# B&R Automation Studio project CleanChemi_SiteManagementSystem (part 21)

#### CMD.st
```iecst
ACTION Modbus_CMD_action:

	// --------------------------------------------------------------------
	// Variable Write Commands
	// --------------------------------------------------------------------

	// AS Block 12 - UNIT_ID
	IF gCMD_LR[IdxSkids_LR].Write_UNIT_ID.Send THEN
		MasterConfig_LR[IdxSkids_LR].action_enable[11].single := TRUE;
		gCMD_LR[IdxSkids_LR].Write_UNIT_ID.Send := FALSE;
	END_IF;

	// AS Block 13 - P201_STRT_CMD
	IF gCMD_LR[IdxSkids_LR].Write_P201_STRT_CMD.Send THEN
		MasterConfig_LR[IdxSkids_LR].action_enable[12].single := TRUE;
		gCMD_LR[IdxSkids_LR].Write_P201_STRT_CMD.Send := FALSE;
	END_IF;

	// AS Block 14 - P201_STP_CMD
	IF gCMD_LR[IdxSkids_LR].Write_P201_STP_CMD.Send THEN
		MasterConfig_LR[IdxSkids_LR].action_enable[13].single := TRUE;
		gCMD_LR[IdxSkids_LR].Write_P201_STP_CMD.Send := FALSE;
	END_IF;

	// AS Block 15 - P201_HOA
	IF gCMD_LR[IdxSkids_LR].Write_P201_HOA.Send THEN
		gCMD_LR[IdxSkids_LR].Write_P201_HOA.wP201_HOA := STRING_TO_UINT(gCMD_LR[IdxSkids_LR].Write_P201_HOA.wP201_HOA_String);
		MasterConfig_LR[IdxSkids_LR].action_enable[14].single := TRUE;
		gCMD_LR[IdxSkids_LR].Write_P201_HOA.Send := FALSE;
	ELSIF NOT gVis.Main.Out.DialogOpen THEN
		gCMD_LR[IdxSkids_LR].Write_P201_HOA.wP201_HOA_String := UINT_TO_STRING(gSkid_LR[IdxSkids_LR].Dosing_Pump_201.P201_HOA);
	END_IF;

	// AS Block 16 - P201_PPM
	IF gCMD_LR[IdxSkids_LR].Write_P201_PPM.Send THEN
		gCMD_LR[IdxSkids_LR].Write_P201_PPM.wP201_PPM_SWAPPED := IDEC_REAL_Conv(gCMD_LR[IdxSkids_LR].Write_P201_PPM.wP201_PPM);
		MasterConfig_LR[IdxSkids_LR].action_enable[15].single := TRUE;
		gCMD_LR[IdxSkids_LR].Write_P201_PPM.Send := FALSE;
	END_IF;

	// AS Block 17 - P201_SP
	IF gCMD_LR[IdxSkids_LR].Write_P201_SP.Send THEN
		gCMD_LR[IdxSkids_LR].Write_P201_SP.wP201_SP_SWAPPED := IDEC_REAL_Conv(gCMD_LR[IdxSkids_LR].Write_P201_SP.wP201_SP);
		MasterConfig_LR[IdxSkids_LR].action_enable[16].single := TRUE;
		gCMD_LR[IdxSkids_LR].Write_P201_SP.Send := FALSE;
	END_IF;

	// AS Block 18 - P202_STRT_CMD
	IF gCMD_LR[IdxSkids_LR].Write_P202_STRT_CMD.Send THEN
		MasterConfig_LR[IdxSkids_LR].action_enable[17].single := TRUE;
		gCMD_LR[IdxSkids_LR].Write_P202_STRT_CMD.Send := FALSE;
	END_IF;

	// AS Block 19 - P202_STP_CMD
	IF gCMD_LR[IdxSkids_LR].Write_P202_STP_CMD.Send THEN
		MasterConfig_LR[IdxSkids_LR].action_enable[18].single := TRUE;
		gCMD_LR[IdxSkids_LR].Write_P202_STP_CMD.Send := FALSE;
	END_IF;

	// AS Block 20 - P202_HOA
	IF gCMD_LR[IdxSkids_LR].Write_P202_HOA.Send THEN
		gCMD_LR[IdxSkids_LR].Write_P202_HOA.wP202_HOA := STRING_TO_UINT(gCMD_LR[IdxSkids_LR].Write_P202_HOA.wP202_HOA_String);
		MasterConfig_LR[IdxSkids_LR].action_enable[19].single := TRUE;
		gCMD_LR[IdxSkids_LR].Write_P202_HOA.Send := FALSE;
	ELSIF NOT gVis.Main.Out.DialogOpen THEN
		gCMD_LR[IdxSkids_LR].Write_P202_HOA.wP202_HOA_String := UINT_TO_STRING(gSkid_LR[IdxSkids_LR].Dosing_Pump_202.P202_HOA);
	END_IF;

	// AS Block 21 - P202_PPM
	IF gCMD_LR[IdxSkids_LR].Write_P202_PPM.Send THEN
		gCMD_LR[IdxSkids_LR].Write_P202_PPM.wP202_PPM_SWAPPED := IDEC_REAL_Conv(gCMD_LR[IdxSkids_LR].Write_P202_PPM.wP202_PPM);
		MasterConfig_LR[IdxSkids_LR].action_enable[20].single := TRUE;
		gCMD_LR[IdxSkids_LR].Write_P202_PPM.Send := FALSE;
	END_IF;

	// AS Block 22 - P202_SP
	IF gCMD_LR[IdxSkids_LR].Write_P202_SP.Send THEN
		gCMD_LR[IdxSkids_LR].Write_P202_SP.wP202_SP_SWAPPED := IDEC_REAL_Conv(gCMD_LR[IdxSkids_LR].Write_P202_SP.wP202_SP);
		MasterConfig_LR[IdxSkids_LR].action_enable[21].single := TRUE;
		gCMD_LR[IdxSkids_LR].Write_P202_SP.Send := FALSE;
	END_IF;

	// AS Block 23 - P203_STRT_CMD
	IF gCMD_LR[IdxSkids_LR].Write_P203_STRT_CMD.Send THEN
		MasterConfig_LR[IdxSkids_LR].action_enable[22].single := TRUE;
		gCMD_LR[IdxSkids_LR].Write_P203_STRT_CMD.Send := FALSE;
	END_IF;

	// AS Block 24 - P203_STP_CMD
	IF gCMD_LR[IdxSkids_LR].Write_P203_STP_CMD.Send THEN
		MasterConfig_LR[IdxSkids_LR].action_enable[23].single := TRUE;
		gCMD_LR[IdxSkids_LR].Write_P203_STP_CMD.Send := FALSE;
	END_IF;

	// AS Block 25 - P203_HOA
	IF gCMD_LR[IdxSkids_LR].Write_P203_HOA.Send THEN
		gCMD_LR[IdxSkids_LR].Write_P203_HOA.wP203_HOA := STRING_TO_UINT(gCMD_LR[IdxSkids_LR].Write_P203_HOA.wP203_HOA_String);
		MasterConfig_LR[IdxSkids_LR].action_enable[24].single := TRUE;
		gCMD_LR[IdxSkids_LR].Write_P203_HOA.Send := FALSE;
	ELSIF NOT gVis.Main.Out.DialogOpen THEN
		gCMD_LR[IdxSkids_LR].Write_P203_HOA.wP203_HOA_String := UINT_TO_STRING(gSkid_LR[IdxSkids_LR].Dosing_Pump_203.P203_HOA);
	END_IF;

	// AS Block 26 - P203_PPM
	IF gCMD_LR[IdxSkids_LR].Write_P203_PPM.Send THEN
		gCMD_LR[IdxSkids_LR].Write_P203_PPM.wP203_PPM_SWAPPED := IDEC_REAL_Conv(gCMD_LR[IdxSkids_LR].Write_P203_PPM.wP203_PPM);
		MasterConfig_LR[IdxSkids_LR].action_enable[25].single := TRUE;
		gCMD_LR[IdxSkids_LR].Write_P203_PPM.Send := FALSE;
	END_IF;

	// AS Block 27 - P203_SP
	IF gCMD_LR[IdxSkids_LR].Write_P203_SP.Send THEN
		gCMD_LR[IdxSkids_LR].Write_P203_SP.wP203_SP_SWAPPED := IDEC_REAL_Conv(gCMD_LR[IdxSkids_LR].Write_P203_SP.wP203_SP);
		MasterConfig_LR[IdxSkids_LR].action_enable[26].single := TRUE;
		gCMD_LR[IdxSkids_LR].Write_P203_SP.Send := FALSE;
	END_IF;

	// AS Block 28 - EFF_1
	IF gCMD_LR[IdxSkids_LR].Write_EFF_1.Send THEN
		gCMD_LR[IdxSkids_LR].Write_EFF_1.wEFF_1_SWAPPED := IDEC_REAL_Conv(gCMD_LR[IdxSkids_LR].Write_EFF_1.wEFF_1);
		MasterConfig_LR[IdxSkids_LR].action_enable[27].single := TRUE;
		gCMD_LR[IdxSkids_LR].Write_EFF_1.Send := FALSE;
	END_IF;

	// AS Block 29 - EFF_2
	IF gCMD_LR[IdxSkids_LR].Write_EFF_2.Send THEN
		gCMD_LR[IdxSkids_LR].Write_EFF_2.wEFF_2_SWAPPED := IDEC_REAL_Conv(gCMD_LR[IdxSkids_LR].Write_EFF_2.wEFF_2);
		MasterConfig_LR[IdxSkids_LR].action_enable[28].single := TRUE;
		gCMD_LR[IdxSkids_LR].Write_EFF_2.Send := FALSE;
	END_IF;

	// AS Block 30 - NAOH_TO_H2O2
	IF gCMD_LR[IdxSkids_LR].Write_NAOH_TO_H2O2.Send THEN
		gCMD_LR[IdxSkids_LR].Write_NAOH_TO_H2O2.wNAOH_TO_H2O2_SWAPPED := IDEC_REAL_Conv(gCMD_LR[IdxSkids_LR].Write_NAOH_TO_H2O2.wNAOH_TO_H2O2);
		MasterConfig_LR[IdxSkids_LR].action_enable[29].single := TRUE;
		gCMD_LR[IdxSkids_LR].Write_NAOH_TO_H2O2.Send := FALSE;
	END_IF;

	// AS Block 31 - TRI_TO_H2O2
	IF gCMD_LR[IdxSkids_LR].Write_TRI_TO_H2O2.Send THEN
		gCMD_LR[IdxSkids_LR].Write_TRI_TO_H2O2.wTRI_TO_H2O2_SWAPPED := IDEC_REAL_Conv(gCMD_LR[IdxSkids_LR].Write_TRI_TO_H2O2.wTRI_TO_H2O2);
		MasterConfig_LR[IdxSkids_LR].action_enable[30].single := TRUE;
		gCMD_LR[IdxSkids_LR].Write_TRI_TO_H2O2.Send := FALSE;
	END_IF;

	// AS Block 32 - PMAX_HOA
	IF gCMD_LR[IdxSkids_LR].Write_PMAX_HOA.Send THEN
		gCMD_LR[IdxSkids_LR].Write_PMAX_HOA.wPMAX_HOA := STRING_TO_UINT(gCMD_LR[IdxSkids_LR].Write_PMAX_HOA.wPMAX_HOA_String);
		MasterConfig_LR[IdxSkids_LR].action_enable[31].single := TRUE;
		gCMD_LR[IdxSkids_LR].Write_PMAX_HOA.Send := FALSE;
	ELSIF NOT gVis.Main.Out.DialogOpen THEN
		gCMD_LR[IdxSkids_LR].Write_PMAX_HOA.wPMAX_HOA_String := UINT_TO_STRING(gSkid_LR[IdxSkids_LR].Pmax_General_Variables.PMAX_HOA);
	END_IF;

	// AS Block 33 - PMAX_CONC
	IF gCMD_LR[IdxSkids_LR].Write_PMAX_CONC.Send THEN
		gCMD_LR[IdxSkids_LR].Write_PMAX_CONC.wPMAX_CONC_SWAPPED := IDEC_REAL_Conv(gCMD_LR[IdxSkids_LR].Write_PMAX_CONC.wPMAX_CONC);
		MasterConfig_LR[IdxSkids_LR].action_enable[32].single := TRUE;
		gCMD_LR[IdxSkids_LR].Write_PMAX_CONC.Send := FALSE;
	END_IF;

	// AS Block 34 - HP_CONC
	IF gCMD_LR[IdxSkids_LR].Write_HP_CONC.Send THEN
		gCMD_LR[IdxSkids_LR].Write_HP_CONC.wHP_CONC_SWAPPED := IDEC_REAL_Conv(gCMD_LR[IdxSkids_LR].Write_HP_CONC.wHP_CONC);
		MasterConfig_LR[IdxSkids_LR].action_enable[33].single := TRUE;
		gCMD_LR[IdxSkids_LR].Write_HP_CONC.Send := FALSE;
	END_IF;

	// AS Block 35 - NAOH_CONC
	IF gCMD_LR[IdxSkids_LR].Write_NAOH_CONC.Send THEN
		gCMD_LR[IdxSkids_LR].Write_NAOH_CONC.wNAOH_CONC_SWAPPED := IDEC_REAL_Conv(gCMD_LR[IdxSkids_LR].Write_NAOH_CONC.wNAOH_CONC);
		MasterConfig_LR[IdxSkids_LR].action_enable[34].single := TRUE;
		gCMD_LR[IdxSkids_LR].Write_NAOH_CONC.Send := FALSE;
	END_IF;

	// AS Block 36 - P101_STRT_CMD
	IF gCMD_LR[IdxSkids_LR].Write_P101_STRT_CMD.Send THEN
		MasterConfig_LR[IdxSkids_LR].action_enable[35].single := TRUE;
		gCMD_LR[IdxSkids_LR].Write_P101_STRT_CMD.Send := FALSE;
	END_IF;

	// AS Block 37 - P101_STP_CMD
	IF gCMD_LR[IdxSkids_LR].Write_P101_STP_CMD.Send THEN
		MasterConfig_LR[IdxSkids_LR].action_enable[36].single := TRUE;
		gCMD_LR[IdxSkids_LR].Write_P101_STP_CMD.Send := FALSE;
	END_IF;

	// AS Block 38 - P101_SP
	IF gCMD_LR[IdxSkids_LR].Write_P101_SP.Send THEN
		gCMD_LR[IdxSkids_LR].Write_P101_SP.wP101_SP_SWAPPED := IDEC_REAL_Conv(gCMD_LR[IdxSkids_LR].Write_P101_SP.wP101_SP);
		MasterConfig_LR[IdxSkids_LR].action_enable[37].single := TRUE;
		gCMD_LR[IdxSkids_LR].Write_P101_SP.Send := FALSE;
	END_IF;

	// AS Block 39 - P102_STRT_CMD
	IF gCMD_LR[IdxSkids_LR].Write_P102_STRT_CMD.Send THEN
		MasterConfig_LR[IdxSkids_LR].action_enable[38].single := TRUE;
		gCMD_LR[IdxSkids_LR].Write_P102_STRT_CMD.Send := FALSE;
	END_IF;

	// AS Block 40 - P102_STP_CMD
	IF gCMD_LR[IdxSkids_LR].Write_P102_STP_CMD.Send THEN
		MasterConfig_LR[IdxSkids_LR].action_enable[39].single := TRUE;
		gCMD_LR[IdxSkids_LR].Write_P102_STP_CMD.Send := FALSE;
	END_IF;

	// AS Block 41 - P102_SP
	IF gCMD_LR[IdxSkids_LR].Write_P102_SP.Send THEN
		gCMD_LR[IdxSkids_LR].Write_P102_SP.wP102_SP_SWAPPED := IDEC_REAL_Conv(gCMD_LR[IdxSkids_LR].Write_P102_SP.wP102_SP);
		MasterConfig_LR[IdxSkids_LR].action_enable[40].single := TRUE;
		gCMD_LR[IdxSkids_LR].Write_P102_SP.Send := FALSE;
	END_IF;

	// AS Block 42 - P103_STRT_CMD
	IF gCMD_LR[IdxSkids_LR].Write_P103_STRT_CMD.Send THEN
		MasterConfig_LR[IdxSkids_LR].action_enable[41].single := TRUE;
		gCMD_LR[IdxSkids_LR].Write_P103_STRT_CMD.Send := FALSE;
	END_IF;

	// AS Block 43 - P103_STP_CMD
	IF gCMD_LR[IdxSkids_LR].Write_P103_STP_CMD.Send THEN
		MasterConfig_LR[IdxSkids_LR].action_enable[42].single := TRUE;
		gCMD_LR[IdxSkids_LR].Write_P103_STP_CMD.Send := FALSE;
	END_IF;

	// AS Block 44 - P103_SP
	IF gCMD_LR[IdxSkids_LR].Write_P103_SP.Send THEN
		gCMD_LR[IdxSkids_LR].Write_P103_SP.wP103_SP_SWAPPED := IDEC_REAL_Conv(gCMD_LR[IdxSkids_LR].Write_P103_SP.wP103_SP);
		MasterConfig_LR[IdxSkids_LR].action_enable[43].single := TRUE;
		gCMD_LR[IdxSkids_LR].Write_P103_SP.Send := FALSE;
	END_IF;

	// AS Block 45 - P104_STRT_CMD
	IF gCMD_LR[IdxSkids_LR].Write_P104_STRT_CMD.Send THEN
		MasterConfig_LR[IdxSkids_LR].action_enable[44].single := TRUE;
		gCMD_LR[IdxSkids_LR].Write_P103_STRT_CMD.Send := FALSE;
	END_IF;

	// AS Block 46 - P104_STP_CMD
	IF gCMD_LR[IdxSkids_LR].Write_P104_STP_CMD.Send THEN
		MasterConfig_LR[IdxSkids_LR].action_enable[45].single := TRUE;
		gCMD_LR[IdxSkids_LR].Write_P104_STP_CMD.Send := FALSE;
	END_IF;

	// AS Block 47 - P104_SP
	IF gCMD_LR[IdxSkids_LR].Write_P104_SP.Send THEN
		gCMD_LR[IdxSkids_LR].Write_P104_SP.wP104_SP_SWAPPED := IDEC_REAL_Conv(gCMD_LR[IdxSkids_LR].Write_P104_SP.wP104_SP);
		MasterConfig_LR[IdxSkids_LR].action_enable[46].single := TRUE;
		gCMD_LR[IdxSkids_LR].Write_P104_SP.Send := FALSE;
	END_IF;

	// AS Block 48 is a READ block

	// AS Block 49 - LOCK_CMD
	IF gCMD_LR[IdxSkids_LR].Write_LOCK_CMD.Send THEN
		MasterConfig_LR[IdxSkids_LR].action_enable[48].single := TRUE;
		gCMD_LR[IdxSkids_LR].Write_LOCK_CMD.Send := FALSE;
	END_IF;

	// AS Block 50 - UNLOCK_CMD
	IF gCMD_LR[IdxSkids_LR].Write_UNLOCK_CMD.Send THEN
		MasterConfig_LR[IdxSkids_LR].action_enable[49].single := TRUE;
		gCMD_LR[IdxSkids_LR].Write_UNLOCK_CMD.Send := FALSE;
	END_IF;

	// AS Block 51 - FI301_SIM_CMD
	IF gCMD_LR[IdxSkids_LR].Write_FI301_SIM_CMD.Send THEN
		MasterConfig_LR[IdxSkids_LR].action_enable[50].single := TRUE;
		gCMD_LR[IdxSkids_LR].Write_FI301_SIM_CMD.Send := FALSE;
	END_IF;

	// AS Block 52 - FI301_MEA_CMD
	IF gCMD_LR[IdxSkids_LR].Write_FI301_MEA_CMD.Send THEN
		MasterConfig_LR[IdxSkids_LR].action_enable[51].single := TRUE;
		gCMD_LR[IdxSkids_LR].Write_FI301_MEA_CMD.Send := FALSE;
	END_IF;

	// AS Block 53 - FI301_SIM
	IF gCMD_LR[IdxSkids_LR].Write_FI301_SIM.Send THEN
		gCMD_LR[IdxSkids_LR].Write_FI301_SIM.wFI301_SIM_SWAPPED := IDEC_REAL_Conv(gCMD_LR[IdxSkids_LR].Write_FI301_SIM.wFI301_SIM);
		MasterConfig_LR[IdxSkids_LR].action_enable[52].single := TRUE;
		gCMD_LR[IdxSkids_LR].Write_FI301_SIM.Send := FALSE;
	END_IF;

	// AS Block 54 - FI302_SIM_CMD
	IF gCMD_LR[IdxSkids_LR].Write_FI302_SIM_CMD.Send THEN
		MasterConfig_LR[IdxSkids_LR].action_enable[53].single := TRUE;
		gCMD_LR[IdxSkids_LR].Write_FI302_SIM_CMD.Send := FALSE;
	END_IF;

	// AS Block 55 - FI302_MEA_CMD
	IF gCMD_LR[IdxSkids_LR].Write_FI302_MEA_CMD.Send THEN
		MasterConfig_LR[IdxSkids_LR].action_enable[54].single := TRUE;
		gCMD_LR[IdxSkids_LR].Write_FI302_MEA_CMD.Send := FALSE;
	END_IF;

	// AS Block 56 - FI302_SIM
	IF gCMD_LR[IdxSkids_LR].Write_FI302_SIM.Send THEN
		gCMD_LR[IdxSkids_LR].Write_FI302_SIM.wFI302_SIM_SWAPPED := IDEC_REAL_Conv(gCMD_LR[IdxSkids_LR].Write_FI302_SIM.wFI302_SIM);
		MasterConfig_LR[IdxSkids_LR].action_enable[55].single := TRUE;
		gCMD_LR[IdxSkids_LR].Write_FI302_SIM.Send := FALSE;
	END_IF;

	// AS Block 57 - FI303_SIM_CMD
	IF gCMD_LR[IdxSkids_LR].Write_FI303_SIM_CMD.Send THEN
		MasterConfig_LR[IdxSkids_LR].action_enable[56].single := TRUE;
		gCMD_LR[IdxSkids_LR].Write_FI303_SIM_CMD.Send := FALSE;
	END_IF;

	// AS Block 58 - FI303_MEA_CMD
	IF gCMD_LR[IdxSkids_LR].Write_FI303_MEA_CMD.Send THEN
		MasterConfig_LR[IdxSkids_LR].action_enable[57].single := TRUE;
		gCMD_LR[IdxSkids_LR].Write_FI303_MEA_CMD.Send := FALSE;
	END_IF;

	// AS Block 59 - FI303_SIM
	IF gCMD_LR[IdxSkids_LR].Write_FI303_SIM.Send THEN
		gCMD_LR[IdxSkids_LR].Write_FI303_SIM.wFI303_SIM_SWAPPED := IDEC_REAL_Conv(gCMD_LR[IdxSkids_LR].Write_FI303_SIM.wFI303_SIM);
		MasterConfig_LR[IdxSkids_LR].action_enable[58].single := TRUE;
		gCMD_LR[IdxSkids_LR].Write_FI303_SIM.Send := FALSE;
	END_IF;

	// AS Block 60 - UNIT_ACK - RESET OF CONDITION PERFORMED IN MAIN.ST ALARMS RESET
	IF gVis.Main.In.AckAllAlarms_Skid[IdxSkids_LR] THEN
		MasterConfig_LR[IdxSkids_LR].action_enable[59].single := TRUE;
	END_IF;

	// AS Block 61 IS THE TEXT READ INT BLOCK

	// AS Block 62 - XV101_OPEN_CMD
	IF gCMD_LR[IdxSkids_LR].Write_XV101_OPEN_CMD.Send THEN
		MasterConfig_LR[IdxSkids_LR].action_enable[61].single := TRUE;
		gCMD_LR[IdxSkids_LR].Write_XV101_OPEN_CMD.Send := FALSE;
	END_IF;

	// AS Block 63 - XV102_OPEN_CMD
	IF gCMD_LR[IdxSkids_LR].Write_XV102_OPEN_CMD.Send THEN
		MasterConfig_LR[IdxSkids_LR].action_enable[62].single := TRUE;
		gCMD_LR[IdxSkids_LR].Write_XV102_OPEN_CMD.Send := FALSE;
	END_IF;

	// AS Block 64 - XV103_OPEN_CMD
	IF gCMD_LR[IdxSkids_LR].Write_XV103_OPEN_CMD.Send THEN
		MasterConfig_LR[IdxSkids_LR].action_enable[63].single := TRUE;
		gCMD_LR[IdxSkids_LR].Write_XV103_OPEN_CMD.Send := FALSE;
	END_IF;

	// AS Block 65 - XV104_OPEN_CMD
	IF gCMD_LR[IdxSkids_LR].Write_XV104_OPEN_CMD.Send THEN
		MasterConfig_LR[IdxSkids_LR].action_enable[64].single := TRUE;
		gCMD_LR[IdxSkids_LR].Write_XV104_OPEN_CMD.Send := FALSE;
	END_IF;

	// AS Block 66 - XV201_OPEN_CMD
	IF gCMD_LR[IdxSkids_LR].Write_XV201_OPEN_CMD.Send THEN
		MasterConfig_LR[IdxSkids_LR].action_enable[65].single := TRUE;
		gCMD_LR[IdxSkids_LR].Write_XV201_OPEN_CMD.Send := FALSE;
	END_IF;

	// AS Block 67 - XV202_OPEN_CMD
	IF gCMD_LR[IdxSkids_LR].Write_XV202_OPEN_CMD.Send THEN
		MasterConfig_LR[IdxSkids_LR].action_enable[66].single := TRUE;
		gCMD_LR[IdxSkids_LR].Write_XV202_OPEN_CMD.Send := FALSE;
	END_IF;

	// AS Block 68 - XV203_OPEN_CMD
	IF gCMD_LR[IdxSkids_LR].Write_XV203_OPEN_CMD.Send THEN
		MasterConfig_LR[IdxSkids_LR].action_enable[67].single := TRUE;
		gCMD_LR[IdxSkids_LR].Write_XV203_OPEN_CMD.Send := FALSE;
	END_IF;

	// AS Block 69 - AS_USER
	IF gCMD_LR[IdxSkids_LR].Write_AS_USER.Send THEN
		MasterConfig_LR[IdxSkids_LR].action_enable[68].single := TRUE;
		gCMD_LR[IdxSkids_LR].Write_AS_USER.Send := FALSE;
	END_IF;

	// AS Block 70 - AS_ACCESS
	IF gCMD_LR[IdxSkids_LR].Write_AS_ACCESS.Send THEN
		MasterConfig_LR[IdxSkids_LR].action_enable[69].single := TRUE;
		gCMD_LR[IdxSkids_LR].Write_AS_ACCESS.Send := FALSE;
	END_IF;

	// AS Block 71 - TOTALIZER_RESET
	IF gCMD_LR[IdxSkids_LR].Write_TOTALIZER_RESET.Send THEN
		MasterConfig_LR[IdxSkids_LR].action_enable[70].single := TRUE;
		gCMD_LR[IdxSkids_LR].Write_TOTALIZER_RESET.Send := FALSE;
	END_IF;

END_ACTION
```

#### Status.st
```iecst
ACTION Modbus_Status_action:

	ModbusTcpMaster[IdxSkids_LR]();

	// --------------------------------------------------------------------
	// Reset last error information
	// --------------------------------------------------------------------
	IF(reset_error) THEN
		brsmemset(ADR(ModbusTcpMaster[IdxSkids_LR].last_error), 0, 2);
		reset_error := 0;
	END_IF

	// --------------------------------------------------------------------
	// Final Variable Mapping AND Data Conversion - READ
	// --------------------------------------------------------------------

	// force transfer
	// AS Block 1 - 6000 DOSING INT
	gSkid_LR[IdxSkids_LR].Pmax_General_Variables.UNIT_ID := gModbus_LR[IdxSkids_LR].Modbus_PeroxyMAX.Block1_Int[0];
	gSkid_LR[IdxSkids_LR].Pmax_General_Variables.USER_ID := gModbus_LR[IdxSkids_LR].Modbus_PeroxyMAX.Block1_Int[2];
	gSkid_LR[IdxSkids_LR].Pmax_General_Variables.USER_ACCESS := gModbus_LR[IdxSkids_LR].Modbus_PeroxyMAX.Block1_Int[4];
	gSkid_LR[IdxSkids_LR].Pmax_General_Variables.PMAX_HOA := gModbus_LR[IdxSkids_LR].Modbus_PeroxyMAX.Block1_Int[6];
	gSkid_LR[IdxSkids_LR].Pmax_General_Variables.PMAX_STATUS := gModbus_LR[IdxSkids_LR].Modbus_PeroxyMAX.Block1_Int[8];
	gSkid_LR[IdxSkids_LR].Pmax_General_Variables.SCREEN_LOCK := gModbus_LR[IdxSkids_LR].Modbus_PeroxyMAX.Block1_Int[10];

	gSkid_LR[IdxSkids_LR].Pmax_Pump_101.P101_XS := gModbus_LR[IdxSkids_LR].Modbus_PeroxyMAX.Block1_Int[20];
	gSkid_LR[IdxSkids_LR].Sensor_Variables.XV101 := gModbus_LR[IdxSkids_LR].Modbus_PeroxyMAX.Block1_Int[22];
	gSkid_LR[IdxSkids_LR].Sensor_Variables.XV101_ENABLE := gModbus_LR[IdxSkids_LR].Modbus_PeroxyMAX.Block1_Int[24];

	gSkid_LR[IdxSkids_LR].Pmax_Pump_102.P102_XS := gModbus_LR[IdxSkids_LR].Modbus_PeroxyMAX.Block1_Int[32];
	gSkid_LR[IdxSkids_LR].Pmax_Pump_102.P102_WARN := gModbus_LR[IdxSkids_LR].Modbus_PeroxyMAX.Block1_Int[34];
	gSkid_LR[IdxSkids_LR].Pmax_Pump_102.P102_ALARM := gModbus_LR[IdxSkids_LR].Modbus_PeroxyMAX.Block1_Int[36];
	gSkid_LR[IdxSkids_LR].Sensor_Variables.XV102 := gModbus_LR[IdxSkids_LR].Modbus_PeroxyMAX.Block1_Int[38];

	gSkid_LR[IdxSkids_LR].Pmax_Pump_103.P103_XS := gModbus_LR[IdxSkids_LR].Modbus_PeroxyMAX.Block1_Int[48];
	gSkid_LR[IdxSkids_LR].Pmax_Pump_103.P103_WARN := gModbus_LR[IdxSkids_LR].Modbus_PeroxyMAX.Block1_Int[50];
	gSkid_LR[IdxSkids_LR].Pmax_Pump_103.P103_ALARM := gModbus_LR[IdxSkids_LR].Modbus_PeroxyMAX.Block1_Int[52];
	gSkid_LR[IdxSkids_LR].Sensor_Variables.XV103 := gModbus_LR[IdxSkids_LR].Modbus_PeroxyMAX.Block1_Int[54];

	gSkid_LR[IdxSkids_LR].Pmax_Pump_104.P104_XS := gModbus_LR[IdxSkids_LR].Modbus_PeroxyMAX.Block1_Int[64];
	gSkid_LR[IdxSkids_LR].Pmax_Pump_104.P104_WARN := gModbus_LR[IdxSkids_LR].Modbus_PeroxyMAX.Block1_Int[66];
	gSkid_LR[IdxSkids_LR].Pmax_Pump_104.P104_ALARM := gModbus_LR[IdxSkids_LR].Modbus_PeroxyMAX.Block1_Int[68];
	gSkid_LR[IdxSkids_LR].Sensor_Variables.XV104 := gModbus_LR[IdxSkids_LR].Modbus_PeroxyMAX.Block1_Int[70];

	// AS Block 2 - 6000 DOSING INT - SPARE
	//:= gModbus_LR[IdxSkids_LR].Modbus_PeroxyMAX.Block2_Int[0];

	// AS Block 3 - 6000 DOSING REAL
	gSkid_LR[IdxSkids_LR].ConversionRatios.EFF_1:= IDEC_REAL_Conv(gModbus_LR[IdxSkids_LR].Modbus_PeroxyMAX.Block3_Real[0]);
	gSkid_LR[IdxSkids_LR].ConversionRatios.EFF_2:= IDEC_REAL_Conv(gModbus_LR[IdxSkids_LR].Modbus_PeroxyMAX.Block3_Real[1]);
	gSkid_LR[IdxSkids_LR].ConversionRatios.NAOH_TO_H2O2:= IDEC_REAL_Conv(gModbus_LR[IdxSkids_LR].Modbus_PeroxyMAX.Block3_Real[2]);
	gSkid_LR[IdxSkids_LR].ConversionRatios.TRI_TO_H2O2:= IDEC_REAL_Conv(gModbus_LR[IdxSkids_LR].Modbus_PeroxyMAX.Block3_Real[3]);
	gSkid_LR[IdxSkids_LR].ConversionRatios.NAOH_TO_TRI:= IDEC_REAL_Conv(gModbus_LR[IdxSkids_LR].Modbus_PeroxyMAX.Block3_Real[4]);

	gSkid_LR[IdxSkids_LR].Pmax_General_Variables.PMAX_CONC:= IDEC_REAL_Conv(gModbus_LR[IdxSkids_LR].Modbus_PeroxyMAX.Block3_Real[8]);
	gSkid_LR[IdxSkids_LR].Pmax_General_Variables.PMAX_RATE:= IDEC_REAL_Conv(gModbus_LR[IdxSkids_LR].Modbus_PeroxyMAX.Block3_Real[9]);
	gSkid_LR[IdxSkids_LR].Pmax_General_Variables.PMAX_PV:= IDEC_REAL_Conv(gModbus_LR[IdxSkids_LR].Modbus_PeroxyMAX.Block3_Real[10]);
	gSkid_LR[IdxSkids_LR].Pmax_General_Variables.NAOH_CONC:= IDEC_REAL_Conv(gModbus_LR[IdxSkids_LR].Modbus_PeroxyMAX.Block3_Real[11]);
	gSkid_LR[IdxSkids_LR].Pmax_General_Variables.NAOH_CONC_OD:= IDEC_REAL_Conv(gModbus_LR[IdxSkids_LR].Modbus_PeroxyMAX.Block3_Real[12]);
	gSkid_LR[IdxSkids_LR].Pmax_General_Variables.HP_CONC:= IDEC_REAL_Conv(gModbus_LR[IdxSkids_LR].Modbus_PeroxyMAX.Block3_Real[13]);
	gSkid_LR[IdxSkids_LR].Pmax_General_Variables.HP_CONC_OD:= IDEC_REAL_Conv(gModbus_LR[IdxSkids_LR].Modbus_PeroxyMAX.Block3_Real[14]);

	gSkid_LR[IdxSkids_LR].Pmax_Pump_101.P101_SP:= IDEC_REAL_Conv(gModbus_LR[IdxSkids_LR].Modbus_PeroxyMAX.Block3_Real[21]);
	gSkid_LR[IdxSkids_LR].Pmax_Pump_101.P101_PV:= IDEC_REAL_Conv(gModbus_LR[IdxSkids_LR].Modbus_PeroxyMAX.Block3_Real[22]);
	gSkid_LR[IdxSkids_LR].Pmax_Pump_101.P101_OP:= IDEC_REAL_Conv(gModbus_LR[IdxSkids_LR].Modbus_PeroxyMAX.Block3_Real[23]);
	gSkid_LR[IdxSkids_LR].Pmax_Pump_101.P101_FQ:= IDEC_REAL_Conv(gModbus_LR[IdxSkids_LR].Modbus_PeroxyMAX.Block3_Real[24]);
	gSkid_LR[IdxSkids_LR].Pmax_Pump_101.P101_TI:= IDEC_REAL_Conv(gModbus_LR[IdxSkids_LR].Modbus_PeroxyMAX.Block3_Real[25]);
	gSkid_LR[IdxSkids_LR].Pmax_Pump_101.P101_PI:= IDEC_REAL_Conv(gModbus_LR[IdxSkids_LR].Modbus_PeroxyMAX.Block3_Real[26]);
	gSkid_LR[IdxSkids_LR].Pmax_Pump_101.P101_PFI:= IDEC_REAL_Conv(gModbus_LR[IdxSkids_LR].Modbus_PeroxyMAX.Block3_Real[27]);
	gSkid_LR[IdxSkids_LR].Pmax_Pump_101.P101_LS:= IDEC_REAL_Conv(gModbus_LR[IdxSkids_LR].Modbus_PeroxyMAX.Block3_Real[28]);

	gSkid_LR[IdxSkids_LR].Pmax_Pump_101B.P101B_OP:= IDEC_REAL_Conv(gModbus_LR[IdxSkids_LR].Modbus_PeroxyMAX.Block3_Real[35]);
	gSkid_LR[IdxSkids_LR].Pmax_Pump_101B.P101B_PFI:= IDEC_REAL_Conv(gModbus_LR[IdxSkids_LR].Modbus_PeroxyMAX.Block3_Real[36]);
	gSkid_LR[IdxSkids_LR].Pmax_Pump_101B.P101B_SP:= IDEC_REAL_Conv(gModbus_LR[IdxSkids_LR].Modbus_PeroxyMAX.Block3_Real[37]);
	gSkid_LR[IdxSkids_LR].Pmax_Pump_101B.P101B_LS:= IDEC_REAL_Conv(gModbus_LR[IdxSkids_LR].Modbus_PeroxyMAX.Block3_Real[38]);

	gSkid_LR[IdxSkids_LR].Pmax_Pump_102.P102_SP:= IDEC_REAL_Conv(gModbus_LR[IdxSkids_LR].Modbus_PeroxyMAX.Block3_Real[45]);
	gSkid_LR[IdxSkids_LR].Pmax_Pump_102.P102_PV:= IDEC_REAL_Conv(gModbus_LR[IdxSkids_LR].Modbus_PeroxyMAX.Block3_Real[46]);
	gSkid_LR[IdxSkids_LR].Pmax_Pump_102.P102_OP:= IDEC_REAL_Conv(gModbus_LR[IdxSkids_LR].Modbus_PeroxyMAX.Block3_Real[47]);
	gSkid_LR[IdxSkids_LR].Pmax_Pump_102.P102_PFI:= IDEC_REAL_Conv(gModbus_LR[IdxSkids_LR].Modbus_PeroxyMAX.Block3_Real[48]);
	gSkid_LR[IdxSkids_LR].Pmax_Pump_102.P102_FQ:= IDEC_REAL_Conv(gModbus_LR[IdxSkids_LR].Modbus_PeroxyMAX.Block3_Real[49]);
	gSkid_LR[IdxSkids_LR].Pmax_Pump_102.P102_PFQ:= IDEC_REAL_Conv(gModbus_LR[IdxSkids_LR].Modbus_PeroxyMAX.Block3_Real[50]);
	gSkid_LR[IdxSkids_LR].Pmax_Pump_102.P102_PPI:= IDEC_REAL_Conv(gModbus_LR[IdxSkids_LR].Modbus_PeroxyMAX.Block3_Real[51]);
	gSkid_LR[IdxSkids_LR].Pmax_Pump_102.P102_TI:= IDEC_REAL_Conv(gModbus_LR[IdxSkids_LR].Modbus_PeroxyMAX.Block3_Real[52]);
	gSkid_LR[IdxSkids_LR].Pmax_Pump_102.P102_PI:= IDEC_REAL_Conv(gModbus_LR[IdxSkids_LR].Modbus_PeroxyMAX.Block3_Real[53]);
	gSkid_LR[IdxSkids_LR].Pmax_Pump_102.P102_LS:= IDEC_REAL_Conv(gModbus_LR[IdxSkids_LR].Modbus_PeroxyMAX.Block3_Real[54]);

	gSkid_LR[IdxSkids_LR].Pmax_Pump_103.P103_SP:= IDEC_REAL_Conv(gModbus_LR[IdxSkids_LR].Modbus_PeroxyMAX.Block3_Real[59]);
	gSkid_LR[IdxSkids_LR].Pmax_Pump_103.P103_PV:= IDEC_REAL_Conv(gModbus_LR[IdxSkids_LR].Modbus_PeroxyMAX.Block3_Real[60]);
	gSkid_LR[IdxSkids_LR].Pmax_Pump_103.P103_OP:= IDEC_REAL_Conv(gModbus_LR[IdxSkids_LR].Modbus_PeroxyMAX.Block3_Real[61]);
	gSkid_LR[IdxSkids_LR].Pmax_Pump_103.P103_PFI:= IDEC_REAL_Conv(gModbus_LR[IdxSkids_LR].Modbus_PeroxyMAX.Block3_Real[62]);

	// AS Block 4 - 6000 DOSING REAL
	gSkid_LR[IdxSkids_LR].Pmax_Pump_103.P103_FQ:= IDEC_REAL_Conv(gModbus_LR[IdxSkids_LR].Modbus_PeroxyMAX.Block4_Real[0]);
	gSkid_LR[IdxSkids_LR].Pmax_Pump_103.P103_PFQ:= IDEC_REAL_Conv(gModbus_LR[IdxSkids_LR].Modbus_PeroxyMAX.Block4_Real[1]);
	gSkid_LR[IdxSkids_LR].Pmax_Pump_103.P103_PPI:= IDEC_REAL_Conv(gModbus_LR[IdxSkids_LR].Modbus_PeroxyMAX.Block4_Real[2]);
	gSkid_LR[IdxSkids_LR].Pmax_Pump_103.P103_TI:= IDEC_REAL_Conv(gModbus_LR[IdxSkids_LR].Modbus_PeroxyMAX.Block4_Real[3]);
	gSkid_LR[IdxSkids_LR].Pmax_Pump_103.P103_PI:= IDEC_REAL_Conv(gModbus_LR[IdxSkids_LR].Modbus_PeroxyMAX.Block4_Real[4]);
	gSkid_LR[IdxSkids_LR].Pmax_Pump_103.P103_LS:= IDEC_REAL_Conv(gModbus_LR[IdxSkids_LR].Modbus_PeroxyMAX.Block4_Real[5]);

	gSkid_LR[IdxSkids_LR].Pmax_Pump_104.P104_SP:= IDEC_REAL_Conv(gModbus_LR[IdxSkids_LR].Modbus_PeroxyMAX.Block4_Real[10]);
	gSkid_LR[IdxSkids_LR].Pmax_Pump_104.P104_PV:= IDEC_REAL_Conv(gModbus_LR[IdxSkids_LR].Modbus_PeroxyMAX.Block4_Real[11]);
	gSkid_LR[IdxSkids_LR].Pmax_Pump_104.P104_OP:= IDEC_REAL_Conv(gModbus_LR[IdxSkids_LR].Modbus_PeroxyMAX.Block4_Real[12]);
	gSkid_LR[IdxSkids_LR].Pmax_Pump_104.P104_PFI:= IDEC_REAL_Conv(gModbus_LR[IdxSkids_LR].Modbus_PeroxyMAX.Block4_Real[13]);
	gSkid_LR[IdxSkids_LR].Pmax_Pump_104.P104_FQ:= IDEC_REAL_Conv(gModbus_LR[IdxSkids_LR].Modbus_PeroxyMAX.Block4_Real[14]);
	gSkid_LR[IdxSkids_LR].Pmax_Pump_104.P104_PFQ:= IDEC_REAL_Conv(gModbus_LR[IdxSkids_LR].Modbus_PeroxyMAX.Block4_Real[15]);
	gSkid_LR[IdxSkids_LR].Pmax_Pump_104.P104_PPI:= IDEC_REAL_Conv(gModbus_LR[IdxSkids_LR].Modbus_PeroxyMAX.Block4_Real[16]);
	gSkid_LR[IdxSkids_LR].Pmax_Pump_104.P104_PI:= IDEC_REAL_Conv(gModbus_LR[IdxSkids_LR].Modbus_PeroxyMAX.Block4_Real[17]);
	gSkid_LR[IdxSkids_LR].Pmax_Pump_104.P104_LS:= IDEC_REAL_Conv(gModbus_LR[IdxSkids_LR].Modbus_PeroxyMAX.Block4_Real[18]);

	gSkid_LR[IdxSkids_LR].Sensor_Variables.CD101:= IDEC_REAL_Conv(gModbus_LR[IdxSkids_LR].Modbus_PeroxyMAX.Block4_Real[24]);
	gSkid_LR[IdxSkids_LR].Sensor_Variables.CD101_SP:= IDEC_REAL_Conv(gModbus_LR[IdxSkids_LR].Modbus_PeroxyMAX.Block4_Real[25]);
	gSkid_LR[IdxSkids_LR].Sensor_Variables.CD102:= IDEC_REAL_Conv(gModbus_LR[IdxSkids_LR].Modbus_PeroxyMAX.Block4_Real[26]);
	gSkid_LR[IdxSkids_LR].Sensor_Variables.CD102_SP:= IDEC_REAL_Conv(gModbus_LR[IdxSkids_LR].Modbus_PeroxyMAX.Block4_Real[27]);
	gSkid_LR[IdxSkids_LR].Sensor_Variables.CD103:= IDEC_REAL_Conv(gModbus_LR[IdxSkids_LR].Modbus_PeroxyMAX.Block4_Real[28]);
	gSkid_LR[IdxSkids_LR].Sensor_Variables.CD103_SP:= IDEC_REAL_Conv(gModbus_LR[IdxSkids_LR].Modbus_PeroxyMAX.Block4_Real[29]);

	gSkid_LR[IdxSkids_LR].Sensor_Variables.CD101_TI:= IDEC_REAL_Conv(gModbus_LR[IdxSkids_LR].Modbus_PeroxyMAX.Block4_Real[36]);
	gSkid_LR[IdxSkids_LR].Sensor_Variables.CD102_TI:= IDEC_REAL_Conv(gModbus_LR[IdxSkids_LR].Modbus_PeroxyMAX.Block4_Real[37]);
	gSkid_LR[IdxSkids_LR].Sensor_Variables.CD103_TI:= IDEC_REAL_Conv(gModbus_LR[IdxSkids_LR].Modbus_PeroxyMAX.Block4_Real[38]);

	gSkid_LR[IdxSkids_LR].Pmax_General_Variables.HMI_REV_A:= IDEC_REAL_Conv(gModbus_LR[IdxSkids_LR].Modbus_PeroxyMAX.Block4_Real[45]);
	gSkid_LR[IdxSkids_LR].Pmax_General_Variables.HMI_REV_B:= IDEC_REAL_Conv(gModbus_LR[IdxSkids_LR].Modbus_PeroxyMAX.Block4_Real[46]);
	gSkid_LR[IdxSkids_LR].Pmax_General_Variables.PLC_REV_A:= IDEC_REAL_Conv(gModbus_LR[IdxSkids_LR].Modbus_PeroxyMAX.Block4_Real[47]);
	gSkid_LR[IdxSkids_LR].Pmax_General_Variables.PLC_REV_B:= IDEC_REAL_Conv(gModbus_LR[IdxSkids_LR].Modbus_PeroxyMAX.Block4_Real[48]);

	gSkid_LR[IdxSkids_LR].BufferTank.LI200:= IDEC_REAL_Conv(gModbus_LR[IdxSkids_LR].Modbus_PeroxyMAX.Block4_Real[51]);
	gSkid_LR[IdxSkids_LR].BufferTank.LSHH200:= IDEC_REAL_Conv(gModbus_LR[IdxSkids_LR].Modbus_PeroxyMAX.Block4_Real[52]);
	gSkid_LR[IdxSkids_LR].BufferTank.DRAINTIME_SP:= IDEC_REAL_Conv(gModbus_LR[IdxSkids_LR].Modbus_PeroxyMAX.Block4_Real[53]);
	gSkid_LR[IdxSkids_LR].BufferTank.DRAINTIME_PV:= IDEC_REAL_Conv(gModbus_LR[IdxSkids_LR].Modbus_PeroxyMAX.Block4_Real[54]);
	gSkid_LR[IdxSkids_LR].BufferTank.FILLTIME_SP:= IDEC_REAL_Conv(gModbus_LR[IdxSkids_LR].Modbus_PeroxyMAX.Block4_Real[55]);
	gSkid_LR[IdxSkids_LR].BufferTank.FILLTIME_PV:= IDEC_REAL_Conv(gModbus_LR[IdxSkids_LR].Modbus_PeroxyMAX.Block4_Real[56]);

	// AS Block 5 - 6000 DOSING REAL - SPARE
	//:= IDEC_REAL_Conv(gModbus_LR[IdxSkids_LR].Modbus_PeroxyMAX.Block5_Real[0]);

	// AS Block 6 - 7000 DOSING INT
	gSkid_LR[IdxSkids_LR].Pmax_General_Variables.UNIT_ID_DOSE := gModbus_LR[IdxSkids_LR].Modbus_Dosing.Block6_Int[0];

	gSkid_LR[IdxSkids_LR].Dosing_Pump_201.P201_XS := gModbus_LR[IdxSkids_LR].Modbus_Dosing.Block6_Int[6];
	gSkid_LR[IdxSkids_LR].Dosing_Pump_201.P201_HOA := gModbus_LR[IdxSkids_LR].Modbus_Dosing.Block6_Int[8];
	gSkid_LR[IdxSkids_LR].Dosing_Pump_201.P201_CHEM := gModbus_LR[IdxSkids_LR].Modbus_Dosing.Block6_Int[10];
	gSkid_LR[IdxSkids_LR].Dosing_Pump_201.P201_ENABLE := gModbus_LR[IdxSkids_LR].Modbus_Dosing.Block6_Int[12];
	gSkid_LR[IdxSkids_LR].Dosing_Pump_201.P201_ADJ := gModbus_LR[IdxSkids_LR].Modbus_Dosing.Block6_Int[14];
	gSkid_LR[IdxSkids_LR].Dosing_Pump_201.P201_PTYPE := gModbus_LR[IdxSkids_LR].Modbus_Dosing.Block6_Int[16];
	gSkid_LR[IdxSkids_LR].Dosing_Pump_201.P201_WARN := gModbus_LR[IdxSkids_LR].Modbus_Dosing.Block6_Int[18];
	gSkid_LR[IdxSkids_LR].Dosing_Pump_201.P201_ALARM := gModbus_LR[IdxSkids_LR].Modbus_Dosing.Block6_Int[20];
	gSkid_LR[IdxSkids_LR].Sensor_Variables.XV201 := gModbus_LR[IdxSkids_LR].Modbus_Dosing.Block6_Int[22];

	gSkid_LR[IdxSkids_LR].Dosing_Pump_202.P202_XS := gModbus_LR[IdxSkids_LR].Modbus_Dosing.Block6_Int[32];
	gSkid_LR[IdxSkids_LR].Dosing_Pump_202.P202_HOA := gModbus_LR[IdxSkids_LR].Modbus_Dosing.Block6_Int[34];
	gSkid_LR[IdxSkids_LR].Dosing_Pump_202.P202_CHEM := gModbus_LR[IdxSkids_LR].Modbus_Dosing.Block6_Int[36];
	gSkid_LR[IdxSkids_LR].Dosing_Pump_202.P202_ENABLE := gModbus_LR[IdxSkids_LR].Modbus_Dosing.Block6_Int[38];
	gSkid_LR[IdxSkids_LR].Dosing_Pump_202.P202_ADJ := gModbus_LR[IdxSkids_LR].Modbus_Dosing.Block6_Int[40];
	gSkid_LR[IdxSkids_LR].Dosing_Pump_202.P202_WARN := gModbus_LR[IdxSkids_LR].Modbus_Dosing.Block6_Int[42];
	gSkid_LR[IdxSkids_LR].Dosing_Pump_202.P202_ALARM := gModbus_LR[IdxSkids_LR].Modbus_Dosing.Block6_Int[44];
	gSkid_LR[IdxSkids_LR].Sensor_Variables.XV202 := gModbus_LR[IdxSkids_LR].Modbus_Dosing.Block6_Int[46];

	gSkid_LR[IdxSkids_LR].Dosing_Pump_203.P203_XS := gModbus_LR[IdxSkids_LR].Modbus_Dosing.Block6_Int[56];
	gSkid_LR[IdxSkids_LR].Dosing_Pump_203.P203_HOA := gModbus_LR[IdxSkids_LR].Modbus_Dosing.Block6_Int[58];
	gSkid_LR[IdxSkids_LR].Dosing_Pump_203.P203_CHEM := gModbus_LR[IdxSkids_LR].Modbus_Dosing.Block6_Int[60];
	gSkid_LR[IdxSkids_LR].Dosing_Pump_203.P203_ENABLE := gModbus_LR[IdxSkids_LR].Modbus_Dosing.Block6_Int[62];
	gSkid_LR[IdxSkids_LR].Dosing_Pump_203.P203_ADJ := gModbus_LR[IdxSkids_LR].Modbus_Dosing.Block6_Int[64];
	gSkid_LR[IdxSkids_LR].Dosing_Pump_203.P203_WARN := gModbus_LR[IdxSkids_LR].Modbus_Dosing.Block6_Int[66];
	gSkid_LR[IdxSkids_LR].Dosing_Pump_203.P203_ALARM := gModbus_LR[IdxSkids_LR].Modbus_Dosing.Block6_Int[68];
	gSkid_LR[IdxSkids_LR].Sensor_Variables.XV203 := gModbus_LR[IdxSkids_LR].Modbus_Dosing.Block6_Int[70];

	gSkid_LR[IdxSkids_LR].Dosing_Pump_204.P204_XS := gModbus_LR[IdxSkids_LR].Modbus_Dosing.Block6_Int[80];
	gSkid_LR[IdxSkids_LR].Dosing_Pump_204.P204_HOA := gModbus_LR[IdxSkids_LR].Modbus_Dosing.Block6_Int[82];
	gSkid_LR[IdxSkids_LR].Dosing_Pump_204.P204_CHEM := gModbus_LR[IdxSkids_LR].Modbus_Dosing.Block6_Int[84];

	gSkid_LR[IdxSkids_LR].Dosing_Pump_205.P205_XS := gModbus_LR[IdxSkids_LR].Modbus_Dosing.Block6_Int[104];
	gSkid_LR[IdxSkids_LR].Dosing_Pump_205.P205_HOA := gModbus_LR[IdxSkids_LR].Modbus_Dosing.Block6_Int[106];
	gSkid_LR[IdxSkids_LR].Dosing_Pump_205.P205_CHEM := gModbus_LR[IdxSkids_LR].Modbus_Dosing.Block6_Int[108];

	// AS Block 7 - 7000 DOSING INT
	gSkid_LR[IdxSkids_LR].Dosing_Pump_206.P206_XS := gModbus_LR[IdxSkids_LR].Modbus_Dosing.Block7_Int[2];
	gSkid_LR[IdxSkids_LR].Dosing_Pump_206.P206_HOA := gModbus_LR[IdxSkids_LR].Modbus_Dosing.Block7_Int[4];
	gSkid_LR[IdxSkids_LR].Dosing_Pump_206.P206_CHEM := gModbus_LR[IdxSkids_LR].Modbus_Dosing.Block7_Int[6];

	gSkid_LR[IdxSkids_LR].Dosing_Pump_207.P207_XS := gModbus_LR[IdxSkids_LR].Modbus_Dosing.Block7_Int[26];
	gSkid_LR[IdxSkids_LR].Dosing_Pump_207.P207_HOA := gModbus_LR[IdxSkids_LR].Modbus_Dosing.Block7_Int[28];
	gSkid_LR[IdxSkids_LR].Dosing_Pump_207.P207_CHEM := gModbus_LR[IdxSkids_LR].Modbus_Dosing.Block7_Int[30];

	gSkid_LR[IdxSkids_LR].Dosing_Pump_208.P208_XS := gModbus_LR[IdxSkids_LR].Modbus_Dosing.Block7_Int[50];
	gSkid_LR[IdxSkids_LR].Dosing_Pump_208.P208_HOA := gModbus_LR[IdxSkids_LR].Modbus_Dosing.Block7_Int[52];
	gSkid_LR[IdxSkids_LR].Dosing_Pump_208.P208_CHEM := gModbus_LR[IdxSkids_LR].Modbus_Dosing.Block7_Int[54];

	gSkid_LR[IdxSkids_LR].Sensor_Variables.SERNSORS_CONFIG := gModbus_LR[IdxSkids_LR].Modbus_Dosing.Block7_Int[104];

	gSkid_LR[IdxSkids_LR].Sensor_Variables.FI301_MODE := gModbus_LR[IdxSkids_LR].Modbus_Dosing.Block7_Int[118];
	gSkid_LR[IdxSkids_LR].Sensor_Variables.FI302_MODE := gModbus_LR[IdxSkids_LR].Modbus_Dosing.Block7_Int[120];
	gSkid_LR[IdxSkids_LR].Sensor_Variables.FI303_MODE := gModbus_LR[IdxSkids_LR].Modbus_Dosing.Block7_Int[122];
	gSkid_LR[IdxSkids_LR].Sensor_Variables.FI304_MODE := gModbus_LR[IdxSkids_LR].Modbus_Dosing.Block7_Int[124];

	// AS Block 8 - 7000 DOSING REAL
	gSkid_LR[IdxSkids_LR].Dosing_Pump_201.P201_REF_SENSOR := IDEC_REAL_Conv(gModbus_LR[IdxSkids_LR].Modbus_Dosing.Block8_Real[0]);
	gSkid_LR[IdxSkids_LR].Dosing_Pump_201.P201_CONC := IDEC_REAL_Conv(gModbus_LR[IdxSkids_LR].Modbus_Dosing.Block8_Real[1]);
	gSkid_LR[IdxSkids_LR].Dosing_Pump_201.P201_PPM := IDEC_REAL_Conv(gModbus_LR[IdxSkids_LR].Modbus_Dosing.Block8_Real[2]);
	gSkid_LR[IdxSkids_LR].Dosing_Pump_201.P201_APPM := IDEC_REAL_Conv(gModbus_LR[IdxSkids_LR].Modbus_Dosing.Block8_Real[3]);
	gSkid_LR[IdxSkids_LR].Dosing_Pump_201.P201_SP := IDEC_REAL_Conv(gModbus_LR[IdxSkids_LR].Modbus_Dosing.Block8_Real[4]);
	gSkid_LR[IdxSkids_LR].Dosing_Pump_201.P201_PV := IDEC_REAL_Conv(gModbus_LR[IdxSkids_LR].Modbus_Dosing.Block8_Real[5]);
	gSkid_LR[IdxSkids_LR].Dosing_Pump_201.P201_OP := IDEC_REAL_Conv(gModbus_LR[IdxSkids_LR].Modbus_Dosing.Block8_Real[6]);
	gSkid_LR[IdxSkids_LR].Dosing_Pump_201.P201_PFI := IDEC_REAL_Conv(gModbus_LR[IdxSkids_LR].Modbus_Dosing.Block8_Real[7]);
	gSkid_LR[IdxSkids_LR].Dosing_Pump_201.P201_FQ := IDEC_REAL_Conv(gModbus_LR[IdxSkids_LR].Modbus_Dosing.Block8_Real[8]);
	gSkid_LR[IdxSkids_LR].Dosing_Pump_201.P201_PI := IDEC_REAL_Conv(gModbus_LR[IdxSkids_LR].Modbus_Dosing.Block8_Real[9]);
	gSkid_LR[IdxSkids_LR].Dosing_Pump_201.P201_TI := IDEC_REAL_Conv(gModbus_LR[IdxSkids_LR].Modbus_Dosing.Block8_Real[10]);
	gSkid_LR[IdxSkids_LR].Dosing_Pump_201.P201_PFQ := IDEC_REAL_Conv(gModbus_LR[IdxSkids_LR].Modbus_Dosing.Block8_Real[11]);
	gSkid_LR[IdxSkids_LR].Dosing_Pump_201.P201_PPI := IDEC_REAL_Conv(gModbus_LR[IdxSkids_LR].Modbus_Dosing.Block8_Real[12]);
	gSkid_LR[IdxSkids_LR].Dosing_Pump_201.P201_LS := IDEC_REAL_Conv(gModbus_LR[IdxSkids_LR].Modbus_Dosing.Block8_Real[13]);
	gSkid_LR[IdxSkids_LR].Dosing_Pump_201.P201_ASP := IDEC_REAL_Conv(gModbus_LR[IdxSkids_LR].Modbus_Dosing.Block8_Real[14]);

	gSkid_LR[IdxSkids_LR].Dosing_Pump_202.P202_REF_SENSOR := IDEC_REAL_Conv(gModbus_LR[IdxSkids_LR].Modbus_Dosing.Block8_Real[19]);
	gSkid_LR[IdxSkids_LR].Dosing_Pump_202.P202_CONC := IDEC_REAL_Conv(gModbus_LR[IdxSkids_LR].Modbus_Dosing.Block8_Real[20]);
	gSkid_LR[IdxSkids_LR].Dosing_Pump_202.P202_PPM := IDEC_REAL_Conv(gModbus_LR[IdxSkids_LR].Modbus_Dosing.Block8_Real[21]);
	gSkid_LR[IdxSkids_LR].Dosing_Pump_202.P202_APPM := IDEC_REAL_Conv(gModbus_LR[IdxSkids_LR].Modbus_Dosing.Block8_Real[22]);
	gSkid_LR[IdxSkids_LR].Dosing_Pump_202.P202_SP := IDEC_REAL_Conv(gModbus_LR[IdxSkids_LR].Modbus_Dosing.Block8_Real[23]);
	gSkid_LR[IdxSkids_LR].Dosing_Pump_202.P202_PV := IDEC_REAL_Conv(gModbus_LR[IdxSkids_LR].Modbus_Dosing.Block8_Real[24]);
	gSkid_LR[IdxSkids_LR].Dosing_Pump_202.P202_OP := IDEC_REAL_Conv(gModbus_LR[IdxSkids_LR].Modbus_Dosing.Block8_Real[25]);
	gSkid_LR[IdxSkids_LR].Dosing_Pump_202.P202_PFI := IDEC_REAL_Conv(gModbus_LR[IdxSkids_LR].Modbus_Dosing.Block8_Real[26]);
	gSkid_LR[IdxSkids_LR].Dosing_Pump_202.P202_FQ := IDEC_REAL_Conv(gModbus_LR[IdxSkids_LR].Modbus_Dosing.Block8_Real[27]);
	gSkid_LR[IdxSkids_LR].Dosing_Pump_202.P202_PI := IDEC_REAL_Conv(gModbus_LR[IdxSkids_LR].Modbus_Dosing.Block8_Real[28]);
	gSkid_LR[IdxSkids_LR].Dosing_Pump_202.P202_TI := IDEC_REAL_Conv(gModbus_LR[IdxSkids_LR].Modbus_Dosing.Block8_Real[29]);
	gSkid_LR[IdxSkids_LR].Dosing_Pump_202.P202_PFQ := IDEC_REAL_Conv(gModbus_LR[IdxSkids_LR].Modbus_Dosing.Block8_Real[30]);
	gSkid_LR[IdxSkids_LR].Dosing_Pump_202.P202_PPI := IDEC_REAL_Conv(gModbus_LR[IdxSkids_LR].Modbus_Dosing.Block8_Real[31]);
	gSkid_LR[IdxSkids_LR].Dosing_Pump_202.P202_LS := IDEC_REAL_Conv(gModbus_LR[IdxSkids_LR].Modbus_Dosing.Block8_Real[32]);
	gSkid_LR[IdxSkids_LR].Dosing_Pump_202.P202_ASP := IDEC_REAL_Conv(gModbus_LR[IdxSkids_LR].Modbus_Dosing.Block8_Real[33]);

	gSkid_LR[IdxSkids_LR].Dosing_Pump_203.P203_REF_SENSOR := IDEC_REAL_Conv(gModbus_LR[IdxSkids_LR].Modbus_Dosing.Block8_Real[38]);
	gSkid_LR[IdxSkids_LR].Dosing_Pump_203.P203_CONC := IDEC_REAL_Conv(gModbus_LR[IdxSkids_LR].Modbus_Dosing.Block8_Real[39]);
	gSkid_LR[IdxSkids_LR].Dosing_Pump_203.P203_PPM := IDEC_REAL_Conv(gModbus_LR[IdxSkids_LR].Modbus_Dosing.Block8_Real[40]);
	gSkid_LR[IdxSkids_LR].Dosing_Pump_203.P203_APPM := IDEC_REAL_Conv(gModbus_LR[IdxSkids_LR].Modbus_Dosing.Block8_Real[41]);
	gSkid_LR[IdxSkids_LR].Dosing_Pump_203.P203_SP := IDEC_REAL_Conv(gModbus_LR[IdxSkids_LR].Modbus_Dosing.Block8_Real[42]);
	gSkid_LR[IdxSkids_LR].Dosing_Pump_203.P203_PV := IDEC_REAL_Conv(gModbus_LR[IdxSkids_LR].Modbus_Dosing.Block8_Real[43]);
	gSkid_LR[IdxSkids_LR].Dosing_Pump_203.P203_OP := IDEC_REAL_Conv(gModbus_LR[IdxSkids_LR].Modbus_Dosing.Block8_Real[44]);
	gSkid_LR[IdxSkids_LR].Dosing_Pump_203.P203_PFI := IDEC_REAL_Conv(gModbus_LR[IdxSkids_LR].Modbus_Dosing.Block8_Real[45]);
	gSkid_LR[IdxSkids_LR].Dosing_Pump_203.P203_FQ := IDEC_REAL_Conv(gModbus_LR[IdxSkids_LR].Modbus_Dosing.Block8_Real[46]);
	gSkid_LR[IdxSkids_LR].Dosing_Pump_203.P203_PI := IDEC_REAL_Conv(gModbus_LR[IdxSkids_LR].Modbus_Dosing.Block8_Real[47]);
	gSkid_LR[IdxSkids_LR].Dosing_Pump_203.P203_TI := IDEC_REAL_Conv(gModbus_LR[IdxSkids_LR].Modbus_Dosing.Block8_Real[48]);
	gSkid_LR[IdxSkids_LR].Dosing_Pump_203.P203_PFQ := IDEC_REAL_Conv(gModbus_LR[IdxSkids_LR].Modbus_Dosing.Block8_Real[49]);
	gSkid_LR[IdxSkids_LR].Dosing_Pump_203.P203_PPI := IDEC_REAL_Conv(gModbus_LR[IdxSkids_LR].Modbus_Dosing.Block8_Real[50]);
	gSkid_LR[IdxSkids_LR].Dosing_Pump_203.P203_LS := IDEC_REAL_Conv(gModbus_LR[IdxSkids_LR].Modbus_Dosing.Block8_Real[51]);
	gSkid_LR[IdxSkids_LR].Dosing_Pump_203.P203_ASP := IDEC_REAL_Conv(gModbus_LR[IdxSkids_LR].Modbus_Dosing.Block8_Real[52]);

	gSkid_LR[IdxSkids_LR].Dosing_Pump_204.P204_REF_SENSOR := IDEC_REAL_Conv(gModbus_LR[IdxSkids_LR].Modbus_Dosing.Block8_Real[57]);
	gSkid_LR[IdxSkids_LR].Dosing_Pump_204.P204_CONC := IDEC_REAL_Conv(gModbus_LR[IdxSkids_LR].Modbus_Dosing.Block8_Real[58]);
	gSkid_LR[IdxSkids_LR].Dosing_Pump_204.P204_PPM := IDEC_REAL_Conv(gModbus_LR[IdxSkids_LR].Modbus_Dosing.Block8_Real[59]);
	gSkid_LR[IdxSkids_LR].Dosing_Pump_204.P204_APPM := IDEC_REAL_Conv(gModbus_LR[IdxSkids_LR].Modbus_Dosing.Block8_Real[60]);
	gSkid_LR[IdxSkids_LR].Dosing_Pump_204.P204_SP := IDEC_REAL_Conv(gModbus_LR[IdxSkids_LR].Modbus_Dosing.Block8_Real[61]);
	gSkid_LR[IdxSkids_LR].Dosing_Pump_204.P204_PV := IDEC_REAL_Conv(gModbus_LR[IdxSkids_LR].Modbus_Dosing.Block8_Real[62]);

	// AS Block 9 - 7000 DOSING REAL
	gSkid_LR[IdxSkids_LR].Dosing_Pump_204.P204_OP := IDEC_REAL_Conv(gModbus_LR[IdxSkids_LR].Modbus_Dosing.Block9_Real[0]);
	gSkid_LR[IdxSkids_LR].Dosing_Pump_204.P204_PFI := IDEC_REAL_Conv(gModbus_LR[IdxSkids_LR].Modbus_Dosing.Block9_Real[1]);
	gSkid_LR[IdxSkids_LR].Dosing_Pump_204.P204_FQ := IDEC_REAL_Conv(gModbus_LR[IdxSkids_LR].Modbus_Dosing.Block9_Real[2]);
	gSkid_LR[IdxSkids_LR].Dosing_Pump_204.P204_PI := IDEC_REAL_Conv(gModbus_LR[IdxSkids_LR].Modbus_Dosing.Block9_Real[3]);
	gSkid_LR[IdxSkids_LR].Dosing_Pump_204.P204_TI := IDEC_REAL_Conv(gModbus_LR[IdxSkids_LR].Modbus_Dosing.Block9_Real[4]);
	gSkid_LR[IdxSkids_LR].Dosing_Pump_204.P204_PFQ := IDEC_REAL_Conv(gModbus_LR[IdxSkids_LR].Modbus_Dosing.Block9_Real[5]);
	gSkid_LR[IdxSkids_LR].Dosing_Pump_204.P204_PPI := IDEC_REAL_Conv(gModbus_LR[IdxSkids_LR].Modbus_Dosing.Block9_Real[6]);
	gSkid_LR[IdxSkids_LR].Dosing_Pump_204.P204_LS := IDEC_REAL_Conv(gModbus_LR[IdxSkids_LR].Modbus_Dosing.Block9_Real[7]);

	gSkid_LR[IdxSkids_LR].Dosing_Pump_205.P205_REF_SENSOR := IDEC_REAL_Conv(gModbus_LR[IdxSkids_LR].Modbus_Dosing.Block9_Real[13]);
	gSkid_LR[IdxSkids_LR].Dosing_Pump_205.P205_CONC := IDEC_REAL_Conv(gModbus_LR[IdxSkids_LR].Modbus_Dosing.Block9_Real[14]);
	gSkid_LR[IdxSkids_LR].Dosing_Pump_205.P205_PPM := IDEC_REAL_Conv(gModbus_LR[IdxSkids_LR].Modbus_Dosing.Block9_Real[15]);
	gSkid_LR[IdxSkids_LR].Dosing_Pump_205.P205_APPM := IDEC_REAL_Conv(gModbus_LR[IdxSkids_LR].Modbus_Dosing.Block9_Real[16]);
	gSkid_LR[IdxSkids_LR].Dosing_Pump_205.P205_SP := IDEC_REAL_Conv(gModbus_LR[IdxSkids_LR].Modbus_Dosing.Block9_Real[17]);
	gSkid_LR[IdxSkids_LR].Dosing_Pump_205.P205_PV := IDEC_REAL_Conv(gModbus_LR[IdxSkids_LR].Modbus_Dosing.Block9_Real[18]);
	gSkid_LR[IdxSkids_LR].Dosing_Pump_205.P205_OP := IDEC_REAL_Conv(gModbus_LR[IdxSkids_LR].Modbus_Dosing.Block9_Real[19]);
	gSkid_LR[IdxSkids_LR].Dosing_Pump_205.P205_PFI := IDEC_REAL_Conv(gModbus_LR[IdxSkids_LR].Modbus_Dosing.Block9_Real[20]);
	gSkid_LR[IdxSkids_LR].Dosing_Pump_205.P205_FQ := IDEC_REAL_Conv(gModbus_LR[IdxSkids_LR].Modbus_Dosing.Block9_Real[21]);
	gSkid_LR[IdxSkids_LR].Dosing_Pump_205.P205_PI := IDEC_REAL_Conv(gModbus_LR[IdxSkids_LR].Modbus_Dosing.Block9_Real[22]);
	gSkid_LR[IdxSkids_LR].Dosing_Pump_205.P205_TI := IDEC_REAL_Conv(gModbus_LR[IdxSkids_LR].Modbus_Dosing.Block9_Real[23]);
	gSkid_LR[IdxSkids_LR].Dosing_Pump_205.P205_PFQ := IDEC_REAL_Conv(gModbus_LR[IdxSkids_LR].Modbus_Dosing.Block9_Real[24]);
	gSkid_LR[IdxSkids_LR].Dosing_Pump_205.P205_PPI := IDEC_REAL_Conv(gModbus_LR[IdxSkids_LR].Modbus_Dosing.Block9_Real[25]);
	gSkid_LR[IdxSkids_LR].Dosing_Pump_205.P205_LS := IDEC_REAL_Conv(gModbus_LR[IdxSkids_LR].Modbus_Dosing.Block9_Real[26]);

	gSkid_LR[IdxSkids_LR].Dosing_Pump_206.P206_REF_SENSOR := IDEC_REAL_Conv(gModbus_LR[IdxSkids_LR].Modbus_Dosing.Block9_Real[32]);
	gSkid_LR[IdxSkids_LR].Dosing_Pump_206.P206_CONC := IDEC_REAL_Conv(gModbus_LR[IdxSkids_LR].Modbus_Dosing.Block9_Real[33]);
	gSkid_LR[IdxSkids_LR].Dosing_Pump_206.P206_PPM := IDEC_REAL_Conv(gModbus_LR[IdxSkids_LR].Modbus_Dosing.Block9_Real[34]);
	gSkid_LR[IdxSkids_LR].Dosing_Pump_206.P206_APPM := IDEC_REAL_Conv(gModbus_LR[IdxSkids_LR].Modbus_Dosing.Block9_Real[35]);
	gSkid_LR[IdxSkids_LR].Dosing_Pump_206.P206_SP := IDEC_REAL_Conv(gModbus_LR[IdxSkids_LR].Modbus_Dosing.Block9_Real[36]);
	gSkid_LR[IdxSkids_LR].Dosing_Pump_206.P206_PV := IDEC_REAL_Conv(gModbus_LR[IdxSkids_LR].Modbus_Dosing.Block9_Real[37]);
	gSkid_LR[IdxSkids_LR].Dosing_Pump_206.P206_OP := IDEC_REAL_Conv(gModbus_LR[IdxSkids_LR].Modbus_Dosing.Block9_Real[38]);
	gSkid_LR[IdxSkids_LR].Dosing_Pump_206.P206_PFI := IDEC_REAL_Conv(gModbus_LR[IdxSkids_LR].Modbus_Dosing.Block9_Real[39]);
	gSkid_LR[IdxSkids_LR].Dosing_Pump_206.P206_FQ := IDEC_REAL_Conv(gModbus_LR[IdxSkids_LR].Modbus_Dosing.Block9_Real[40]);
	gSkid_LR[IdxSkids_LR].Dosing_Pump_206.P206_PI := IDEC_REAL_Conv(gModbus_LR[IdxSkids_LR].Modbus_Dosing.Block9_Real[41]);
	gSkid_LR[IdxSkids_LR].Dosing_Pump_206.P206_TI := IDEC_REAL_Conv(gModbus_LR[IdxSkids_LR].Modbus_Dosing.Block9_Real[42]);
	gSkid_LR[IdxSkids_LR].Dosing_Pump_206.P206_PFQ := IDEC_REAL_Conv(gModbus_LR[IdxSkids_LR].Modbus_Dosing.Block9_Real[43]);
	gSkid_LR[IdxSkids_LR].Dosing_Pump_206.P206_PPI := IDEC_REAL_Conv(gModbus_LR[IdxSkids_LR].Modbus_Dosing.Block9_Real[44]);
	gSkid_LR[IdxSkids_LR].Dosing_Pump_206.P206_LS := IDEC_REAL_Conv(gModbus_LR[IdxSkids_LR].Modbus_Dosing.Block9_Real[45]);

	gSkid_LR[IdxSkids_LR].Dosing_Pump_207.P207_REF_SENSOR := IDEC_REAL_Conv(gModbus_LR[IdxSkids_LR].Modbus_Dosing.Block9_Real[51]);
	gSkid_LR[IdxSkids_LR].Dosing_Pump_207.P207_CONC := IDEC_REAL_Conv(gModbus_LR[IdxSkids_LR].Modbus_Dosing.Block9_Real[52]);
	gSkid_LR[IdxSkids_LR].Dosing_Pump_207.P207_PPM := IDEC_REAL_Conv(gModbus_LR[IdxSkids_LR].Modbus_Dosing.Block9_Real[53]);
	gSkid_LR[IdxSkids_LR].Dosing_Pump_207.P207_APPM := IDEC_REAL_Conv(gModbus_LR[IdxSkids_LR].Modbus_Dosing.Block9_Real[54]);
	gSkid_LR[IdxSkids_LR].Dosing_Pump_207.P207_SP := IDEC_REAL_Conv(gModbus_LR[IdxSkids_LR].Modbus_Dosing.Block9_Real[55]);
	gSkid_LR[IdxSkids_LR].Dosing_Pump_207.P207_PV := IDEC_REAL_Conv(gModbus_LR[IdxSkids_LR].Modbus_Dosing.Block9_Real[56]);
	gSkid_LR[IdxSkids_LR].Dosing_Pump_207.P207_OP := IDEC_REAL_Conv(gModbus_LR[IdxSkids_LR].Modbus_Dosing.Block9_Real[57]);
	gSkid_LR[IdxSkids_LR].Dosing_Pump_207.P207_PFI := IDEC_REAL_Conv(gModbus_LR[IdxSkids_LR].Modbus_Dosing.Block9_Real[58]);
	gSkid_LR[IdxSkids_LR].Dosing_Pump_207.P207_FQ := IDEC_REAL_Conv(gModbus_LR[IdxSkids_LR].Modbus_Dosing.Block9_Real[59]);
	gSkid_LR[IdxSkids_LR].Dosing_Pump_207.P207_PI := IDEC_REAL_Conv(gModbus_LR[IdxSkids_LR].Modbus_Dosing.Block9_Real[60]);
	gSkid_LR[IdxSkids_LR].Dosing_Pump_207.P207_TI := IDEC_REAL_Conv(gModbus_LR[IdxSkids_LR].Modbus_Dosing.Block9_Real[61]);
	gSkid_LR[IdxSkids_LR].Dosing_Pump_207.P207_PFQ := IDEC_REAL_Conv(gModbus_LR[IdxSkids_LR].Modbus_Dosing.Block9_Real[62]);

	// AS Block 10 - 7000 DOSING REAL
	gSkid_LR[IdxSkids_LR].Dosing_Pump_207.P207_PPI := IDEC_REAL_Conv(gModbus_LR[IdxSkids_LR].Modbus_Dosing.Block10_Real[0]);
	gSkid_LR[IdxSkids_LR].Dosing_Pump_207.P207_LS := IDEC_REAL_Conv(gModbus_LR[IdxSkids_LR].Modbus_Dosing.Block10_Real[1]);

	gSkid_LR[IdxSkids_LR].Dosing_Pump_208.P208_REF_SENSOR := IDEC_REAL_Conv(gModbus_LR[IdxSkids_LR].Modbus_Dosing.Block10_Real[7]);
	gSkid_LR[IdxSkids_LR].Dosing_Pump_208.P208_CONC := IDEC_REAL_Conv(gModbus_LR[IdxSkids_LR].Modbus_Dosing.Block10_Real[8]);
	gSkid_LR[IdxSkids_LR].Dosing_Pump_208.P208_PPM := IDEC_REAL_Conv(gModbus_LR[IdxSkids_LR].Modbus_Dosing.Block10_Real[9]);
	gSkid_LR[IdxSkids_LR].Dosing_Pump_208.P208_APPM := IDEC_REAL_Conv(gModbus_LR[IdxSkids_LR].Modbus_Dosing.Block10_Real[10]);
	gSkid_LR[IdxSkids_LR].Dosing_Pump_208.P208_SP := IDEC_REAL_Conv(gModbus_LR[IdxSkids_LR].Modbus_Dosing.Block10_Real[11]);
	gSkid_LR[IdxSkids_LR].Dosing_Pump_208.P208_PV := IDEC_REAL_Conv(gModbus_LR[IdxSkids_LR].Modbus_Dosing.Block10_Real[12]);
	gSkid_LR[IdxSkids_LR].Dosing_Pump_208.P208_OP := IDEC_REAL_Conv(gModbus_LR[IdxSkids_LR].Modbus_Dosing.Block10_Real[13]);
	gSkid_LR[IdxSkids_LR].Dosing_Pump_208.P208_PFI := IDEC_REAL_Conv(gModbus_LR[IdxSkids_LR].Modbus_Dosing.Block10_Real[14]);
	gSkid_LR[IdxSkids_LR].Dosing_Pump_208.P208_FQ := IDEC_REAL_Conv(gModbus_LR[IdxSkids_LR].Modbus_Dosing.Block10_Real[15]);
	gSkid_LR[IdxSkids_LR].Dosing_Pump_208.P208_PI := IDEC_REAL_Conv(gModbus_LR[IdxSkids_LR].Modbus_Dosing.Block10_Real[16]);
	gSkid_LR[IdxSkids_LR].Dosing_Pump_208.P208_TI := IDEC_REAL_Conv(gModbus_LR[IdxSkids_LR].Modbus_Dosing.Block10_Real[17]);
	gSkid_LR[IdxSkids_LR].Dosing_Pump_208.P208_PFQ := IDEC_REAL_Conv(gModbus_LR[IdxSkids_LR].Modbus_Dosing.Block10_Real[18]);
	gSkid_LR[IdxSkids_LR].Dosing_Pump_208.P208_PPI := IDEC_REAL_Conv(gModbus_LR[IdxSkids_LR].Modbus_Dosing.Block10_Real[19]);
	gSkid_LR[IdxSkids_LR].Dosing_Pump_208.P208_LS := IDEC_REAL_Conv(gModbus_LR[IdxSkids_LR].Modbus_Dosing.Block10_Real[20]);

	gSkid_LR[IdxSkids_LR].Sensor_Variables.SENSOR301 := IDEC_REAL_Conv(gModbus_LR[IdxSkids_LR].Modbus_Dosing.Block10_Real[26]);
	gSkid_LR[IdxSkids_LR].Sensor_Variables.SENSOR302 := IDEC_REAL_Conv(gModbus_LR[IdxSkids_LR].Modbus_Dosing.Block10_Real[27]);
	gSkid_LR[IdxSkids_LR].Sensor_Variables.SENSOR303 := IDEC_REAL_Conv(gModbus_LR[IdxSkids_LR].Modbus_Dosing.Block10_Real[28]);
	gSkid_LR[IdxSkids_LR].Sensor_Variables.SENSOR304 := IDEC_REAL_Conv(gModbus_LR[IdxSkids_LR].Modbus_Dosing.Block10_Real[29]);

	gSkid_LR[IdxSkids_LR].Sensor_Variables.FI301 := IDEC_REAL_Conv(gModbus_LR[IdxSkids_LR].Modbus_Dosing.Block10_Real[34]);
	gSkid_LR[IdxSkids_LR].Sensor_Variables.FI301_QT := IDEC_REAL_Conv(gModbus_LR[IdxSkids_LR].Modbus_Dosing.Block10_Real[35]);
	gSkid_LR[IdxSkids_LR].Sensor_Variables.FI302 := IDEC_REAL_Conv(gModbus_LR[IdxSkids_LR].Modbus_Dosing.Block10_Real[36]);
	gSkid_LR[IdxSkids_LR].Sensor_Variables.FI302_QT := IDEC_REAL_Conv(gModbus_LR[IdxSkids_LR].Modbus_Dosing.Block10_Real[37]);
	gSkid_LR[IdxSkids_LR].Sensor_Variables.FI303 := IDEC_REAL_Conv(gModbus_LR[IdxSkids_LR].Modbus_Dosing.Block10_Real[38]);
	gSkid_LR[IdxSkids_LR].Sensor_Variables.FI303_QT := IDEC_REAL_Conv(gModbus_LR[IdxSkids_LR].Modbus_Dosing.Block10_Real[39]);
	gSkid_LR[IdxSkids_LR].Sensor_Variables.FI304 := IDEC_REAL_Conv(gModbus_LR[IdxSkids_LR].Modbus_Dosing.Block10_Real[40]);
	gSkid_LR[IdxSkids_LR].Sensor_Variables.FI304_QT := IDEC_REAL_Conv(gModbus_LR[IdxSkids_LR].Modbus_Dosing.Block10_Real[41]);

	// AS Block 11 - 7000 DOSING REAL - SPARE
	//:= IDEC_REAL_Conv(gModbus_LR[IdxSkids_LR].Modbus_Dosing.Block11_Real[0]);

	// AS Block 48 - ALARMS
	gSkid_LR[IdxSkids_LR].Alarms.ALARM_AB1 := gModbus_LR[IdxSkids_LR].Modbus_Alarms.Block48_Int[0];
	gSkid_LR[IdxSkids_LR].Alarms.ALARM_AB2 := gModbus_LR[IdxSkids_LR].Modbus_Alarms.Block48_Int[1];
	gSkid_LR[IdxSkids_LR].Alarms.ALARM_AB3 := gModbus_LR[IdxSkids_LR].Modbus_Alarms.Block48_Int[2];
	gSkid_LR[IdxSkids_LR].Alarms.ALARM_AB4 := gModbus_LR[IdxSkids_LR].Modbus_Alarms.Block48_Int[3];
	gSkid_LR[IdxSkids_LR].Alarms.ALARM_AB5 := gModbus_LR[IdxSkids_LR].Modbus_Alarms.Block48_Int[4];
	gSkid_LR[IdxSkids_LR].Alarms.ALARM_AB6 := gModbus_LR[IdxSkids_LR].Modbus_Alarms.Block48_Int[5];
	gSkid_LR[IdxSkids_LR].Alarms.ALARM_AB7 := gModbus_LR[IdxSkids_LR].Modbus_Alarms.Block48_Int[6];
	gSkid_LR[IdxSkids_LR].Alarms.ALARM_AB8 := gModbus_LR[IdxSkids_LR].Modbus_Alarms.Block48_Int[7];
	gSkid_LR[IdxSkids_LR].Alarms.ALARM_P102 := gModbus_LR[IdxSkids_LR].Modbus_Alarms.Block48_Int[13];
	gSkid_LR[IdxSkids_LR].Alarms.ALARM_P103 := gModbus_LR[IdxSkids_LR].Modbus_Alarms.Block48_Int[14];
	gSkid_LR[IdxSkids_LR].Alarms.ALARM_P104 := gModbus_LR[IdxSkids_LR].Modbus_Alarms.Block48_Int[15];
	gSkid_LR[IdxSkids_LR].Alarms.ALARM_P201 := gModbus_LR[IdxSkids_LR].Modbus_Alarms.Block48_Int[16];
	gSkid_LR[IdxSkids_LR].Alarms.ALARM_P202 := gModbus_LR[IdxSkids_LR].Modbus_Alarms.Block48_Int[17];
	gSkid_LR[IdxSkids_LR].Alarms.ALARM_P203 := gModbus_LR[IdxSkids_LR].Modbus_Alarms.Block48_Int[18];

	// AS Block 61 - DOSING PUMP TEXT
	IDEC_String(ADR(gSkid_LR[IdxSkids_LR].Dosing_Pump_201.P201_TEXT),ADR(gModbus_LR[IdxSkids_LR].Modbus_Dosing.Block61_Int[0]),SIZEOF(gSkid_LR[IdxSkids_LR].Dosing_Pump_201.P201_TEXT),27);
	IDEC_String(ADR(gSkid_LR[IdxSkids_LR].Dosing_Pump_202.P202_TEXT),ADR(gModbus_LR[IdxSkids_LR].Modbus_Dosing.Block61_Int[28]),SIZEOF(gSkid_LR[IdxSkids_LR].Dosing_Pump_202.P202_TEXT),27);
	IDEC_String(ADR(gSkid_LR[IdxSkids_LR].Dosing_Pump_203.P203_TEXT),ADR(gModbus_LR[IdxSkids_LR].Modbus_Dosing.Block61_Int[56]),SIZEOF(gSkid_LR[IdxSkids_LR].Dosing_Pump_203.P203_TEXT),27);

END_ACTION
```
